// TIA Portal V19 export
FUNCTION "Area02_HU_CALL" : Void   // FC167, LAD
TITLE = COIL HANDLING MAIN HU (7,5kW) CALL
// stored: SetENOAutomatically false
   VAR_TEMP
      retval : Int;
      OilTemperature : Real;
      AnalTemperature_Real : Real;
   END_VAR
BEGIN

REGION Network 1: Machine Manager
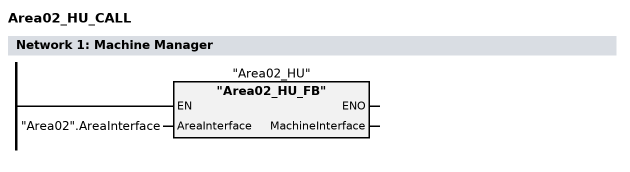
   RUNG wire#powerrail
      "Area02_HU"(AreaInterface := "Area02".AreaInterface, MachineInterface =>)
   END_RUNG
   // the same network as SCL:
   "Area02_HU"(AreaInterface := "Area02".AreaInterface);   // "Area02_HU_FB"
END_REGION
END_FUNCTION
